Omron Sysmac Studio project Benim_Fonk (Sysmac Studio 1.65.0.64007, StandardProject)

# Controller new_Controller_0: NX1P2-1040DT1 version 1.69
Task PrimaryTask (priority 4, period or condition 2000): Program0



PROGRAM Program0
VAR
    Scale_Value : REAL;
    Scale_X0 : REAL;
    Scale_Y0 : REAL;
    Scale_X1 : REAL;
    Scale_Y1 : REAL;
    Scale_Out : REAL;
    Lim_Min : REAL;
    Lim_Max : REAL;
    Lim_Out : REAL;
    Analog_Input : REAL;
    InputMin : REAL;
    OutputMin : REAL;
    OutputMax : REAL;
    BasinsDeg : REAL;
    InputMax : REAL;
END_VAR
VAR
    _t1 : BOOL;
END_VAR

(* Section Section0: ladder, written here as Structured Text *)

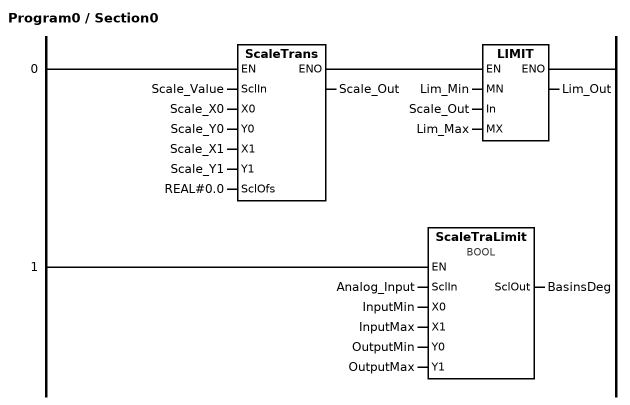
(* Rung 0 *)
Scale_Out := ScaleTrans(SclIn := Scale_Value, X0 := Scale_X0, Y0 := Scale_Y0, X1 := Scale_X1, Y1 := Scale_Y1, SclOfs := REAL#0.0);
Lim_Out := LIMIT(MN := Lim_Min, In := Scale_Out, MX := Lim_Max);
(* Rung 1 *)
_t1 := ScaleTraLimit(SclIn := Analog_Input, X0 := InputMin, X1 := InputMax, Y0 := OutputMin, Y1 := OutputMax, SclOut => BasinsDeg);
END_PROGRAM

FUNCTION ScaleTraLimit : BOOL
VAR
    Scl_Out_Temp : REAL;
END_VAR
VAR_INPUT
    SclIn : REAL;
    X0 : REAL;
    X1 : REAL;
    Y0 : REAL;
    Y1 : REAL;
END_VAR
VAR_OUTPUT
    SclOut : REAL;
END_VAR
(* ladder, written here as Structured Text *)

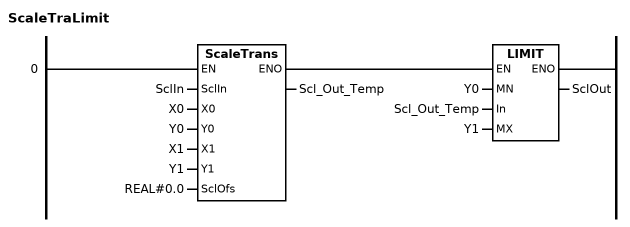
(* Rung 0 *)
Scl_Out_Temp := ScaleTrans(SclIn := SclIn, X0 := X0, Y0 := Y0, X1 := X1, Y1 := Y1, SclOfs := REAL#0.0);
SclOut := LIMIT(MN := Y0, In := Scl_Out_Temp, MX := Y1);
END_FUNCTION